TYPE fbAnalogueValueData :
STRUCT
    ProcessedData : stAnalogueProcessData;
END_STRUCT
END_TYPE

(* stored: Version 1.1.0.1, ProductVersion 3.1.4024.6
   DUT fbAnalogueValueData: Id {0104665c-ddc2-4a4f-9493-a7a2f941dd80} *)
